SYSTEM ece1
  (* Version 1.0, Author, 4DIAC-Consortium *)
  APPLICATION app1
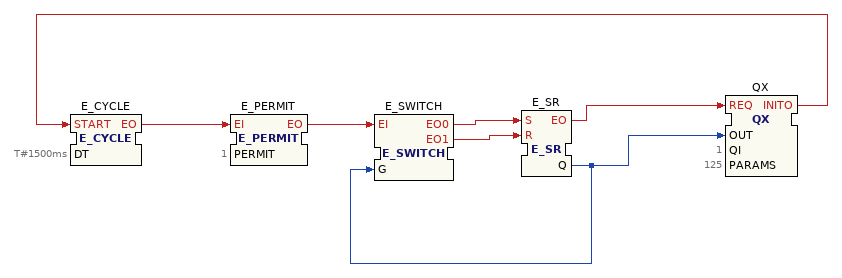
    FBS
      QX : QX(QI := 1, PARAMS := 125);
      E_CYCLE : E_CYCLE(DT := T#1500ms);
      E_SWITCH : E_SWITCH;
      E_SR : E_SR;
      E_PERMIT : E_PERMIT(PERMIT := 1);
    END_FBS
    EVENT_CONNECTIONS
      E_SR.EO TO QX.REQ;
      E_SWITCH.EO0 TO E_SR.S;
      E_SWITCH.EO1 TO E_SR.R;
      QX.INITO TO E_CYCLE.START;
      E_PERMIT.EO TO E_SWITCH.EI;
      E_CYCLE.EO TO E_PERMIT.EI;
    END_CONNECTIONS
    DATA_CONNECTIONS
      E_SR.Q TO QX.OUT;
      E_SR.Q TO E_SWITCH.G;
    END_CONNECTIONS
  END_APPLICATION
  APPLICATION app2
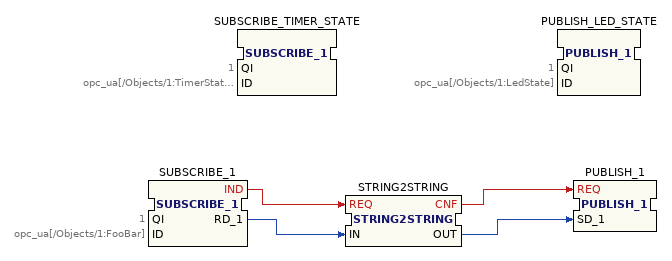
    FBS
      PUBLISH_1 : PUBLISH_1;
      SUBSCRIBE_1 : SUBSCRIBE_1(QI := 1, ID := opc_ua[/Objects/1:FooBar]);
      STRING2STRING : STRING2STRING;
      PUBLISH_LED_STATE : PUBLISH_1(QI := 1, ID := opc_ua[/Objects/1:LedState]);
      SUBSCRIBE_TIMER_STATE : SUBSCRIBE_1(QI := 1, ID := opc_ua[/Objects/1:TimerState]);
    END_FBS
    EVENT_CONNECTIONS
      SUBSCRIBE_1.IND TO STRING2STRING.REQ;
      STRING2STRING.CNF TO PUBLISH_1.REQ;
    END_CONNECTIONS
    DATA_CONNECTIONS
      SUBSCRIBE_1.RD_1 TO STRING2STRING.IN;
      STRING2STRING.OUT TO PUBLISH_1.SD_1;
    END_CONNECTIONS
  END_APPLICATION
  DEVICE RaspberryPI : RaspberryPI(MGR_ID := "localhost:61499")
    {SET_ATTRIBUTE(Profile, HOLOBLOC)}
    RESOURCE EMB_RES : EMB_RES
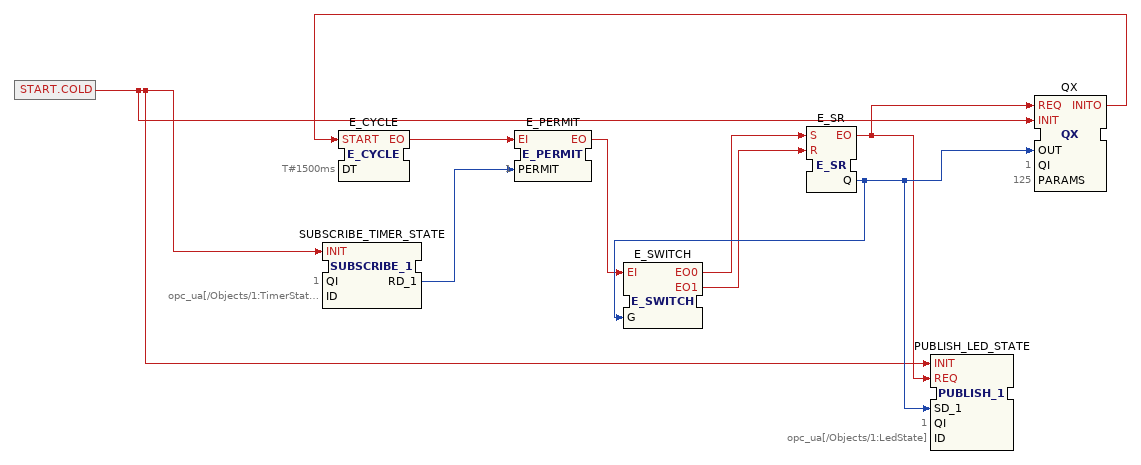
      FBS
        QX : QX(QI := 1, PARAMS := 125);
        E_CYCLE : E_CYCLE(DT := T#1500ms);
        E_SWITCH : E_SWITCH;
        E_SR : E_SR;
        PUBLISH_LED_STATE : PUBLISH_1(QI := 1, ID := opc_ua[/Objects/1:LedState]);
        E_PERMIT : E_PERMIT(PERMIT := 1);
        SUBSCRIBE_TIMER_STATE : SUBSCRIBE_1(QI := 1, ID := opc_ua[/Objects/1:TimerState]);
      END_FBS
      EVENT_CONNECTIONS
        E_SR.EO TO QX.REQ;
        QX.INITO TO E_CYCLE.START;
        E_SWITCH.EO0 TO E_SR.S;
        E_SWITCH.EO1 TO E_SR.R;
        START.COLD TO QX.INIT;
        START.COLD TO PUBLISH_LED_STATE.INIT;
        E_SR.EO TO PUBLISH_LED_STATE.REQ;
        E_CYCLE.EO TO E_PERMIT.EI;
        E_PERMIT.EO TO E_SWITCH.EI;
        START.COLD TO SUBSCRIBE_TIMER_STATE.INIT;
      END_CONNECTIONS
      DATA_CONNECTIONS
        E_SR.Q TO QX.OUT;
        E_SR.Q TO E_SWITCH.G;
        E_SR.Q TO PUBLISH_LED_STATE.SD_1;
        SUBSCRIBE_TIMER_STATE.RD_1 TO E_PERMIT.PERMIT;
      END_CONNECTIONS
    END_RESOURCE
  END_DEVICE
  MAPPINGS
    app1.QX ON RaspberryPI.EMB_RES.QX;
    app1.E_CYCLE ON RaspberryPI.EMB_RES.E_CYCLE;
    app1.E_SWITCH ON RaspberryPI.EMB_RES.E_SWITCH;
    app1.E_SR ON RaspberryPI.EMB_RES.E_SR;
    app2.PUBLISH_LED_STATE ON RaspberryPI.EMB_RES.PUBLISH_LED_STATE;
    app1.E_PERMIT ON RaspberryPI.EMB_RES.E_PERMIT;
    app2.SUBSCRIBE_TIMER_STATE ON RaspberryPI.EMB_RES.SUBSCRIBE_TIMER_STATE;
  END_MAPPINGS
END_SYSTEM
